FUNCTION_BLOCK FB_Roboter_Axis
VAR_INPUT
	bEnable :BOOL;
	bExecute :BOOL;
	rPosition :REAL;
	bRefSens :BOOL;
END_VAR
VAR_OUTPUT
	eState :eBetriebszustand;
END_VAR
VAR
	nState:INT :=0;
	mc_Reset :MC_Reset;
	mc_MoveAbsolute :MC_MoveAbsolute;
	mc_Home :MC_Home;
	mc_Power :MC_Power;
END_VAR
VAR_IN_OUT
	ax :AXIS_REF;
END_VAR

mc_Home(
	Axis:= , 
	Execute:= , 
	Position:= , 
	HomingMode:= , 
	BufferMode:= , 
	Options:= , 
	bCalibrationCam:= , 
	Done=> , 
	Busy=> , 
	Active=> , 
	CommandAborted=> , 
	Error=> , 
	ErrorID=> );
	
mc_MoveAbsolute(
	Axis:= , 
	Execute:= , 
	Position:= , 
	Velocity:= , 
	Acceleration:= , 
	Deceleration:= , 
	Jerk:= , 
	BufferMode:= , 
	Options:= , 
	Done=> , 
	Busy=> , 
	Active=> , 
	CommandAborted=> , 
	Error=> , 
	ErrorID=> );

mc_Power(
	Axis:= , 
	Enable:= , 
	Enable_Positive:= , 
	Enable_Negative:= , 
	Override:= , 
	BufferMode:= , 
	Options:= , 
	Status=> , 
	Busy=> , 
	Error=> , 
	ErrorID=> );
	
mc_Reset(
	Axis:= , 
	Execute:= , 
	Done=> , 
	Busy=> , 
	Error=> , 
	ErrorID=> );

END_FUNCTION_BLOCK

(* stored: Version 1.1.0.1, ProductVersion 3.1.4024.15
   POU FB_Roboter_Axis: Id {bb71503e-a414-410e-8892-e81fc9490a92}, SpecialFunc None *)
